VAR_GLOBAL CONSTANT
	MAX_BUFFER_SIZE : UDINT := 1000;
END_VAR

(* stored: Version 1.1.0.1, ProductVersion 3.1.4024.9
   GVL GVL: Id {2ca9df07-94b3-47a5-a6e5-afe76130c350} *)
